Fanuc TP program (LS listing): UP025.LS

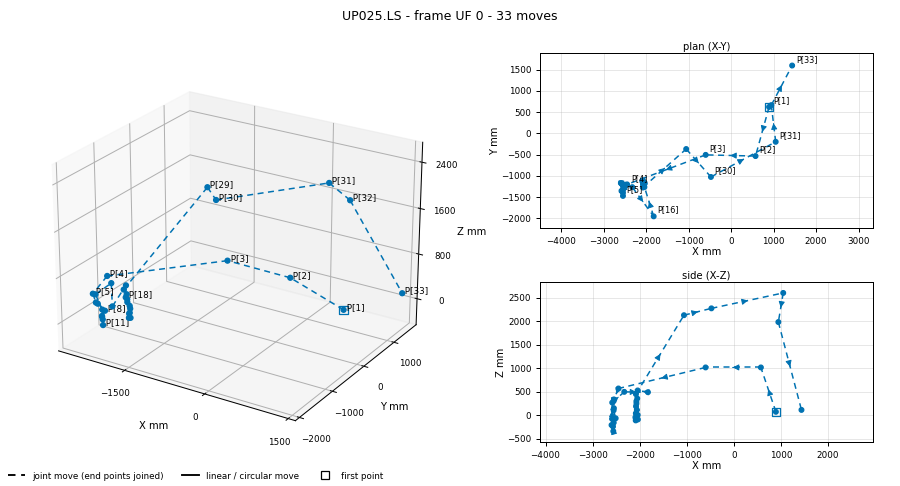
[picture p0: tool path of UP025.LS in frame UF 0, 33 of 33 moves have a stored position in this frame; points joined in program order, loops and branches not executed]
/PROG  UP025
/ATTR
OWNER		= GME;
COMMENT		= "DEPOSITA ST1150";
PROG_SIZE	= 15100;
CREATE		= DATE 03-01-27  TIME 10:40:16;
MODIFIED	= DATE 24-05-04  TIME 16:17:32;
FILE_NAME	= UP025;
VERSION		= 0;
LINE_COUNT	= 60;
MEMORY_SIZE	= 27460;
PROTECT		= READ_WRITE;
TCD:  STACK_SIZE	= 500,
      TASK_PRIORITY	= 50,
      TIME_SLICE	= 0,
      BUSY_LAMP_OFF	= 0,
      ABORT_REQUEST	= 0,
      PAUSE_REQUEST	= 0;
DEFAULT_GROUP	= 1,1,1,1,*;
CONTROL_CODE	= 00000000 00000000;
/APPL
/MN
   1:  UFRAME_NUM=0 ;
   2:  UTOOL_NUM=1 ;
   3:  PAYLOAD[2] ;
   4:  !Apagar Perfil Lib. 74 vs ST1150 ;
   5:  !Apagar Perfil Lib. 73 vs ST1150 ;
   6:  !Encender Anticol. 3 vs 1150R01 ;
   7:  !Encender Anticol. 5 vs 1180R01 ;
   8:J P[1] 100% CNT0 ACC100 TB    0.00sec,P-SPS    ;
      1:  TC_ONLINE (ON) ;
      2:  DO[23]=OFF ;
      3:  TIMER[6]=RESET ;
      4:  TIMER[6]=START ;
      5:  CALL MAKRO050    ;
      6:  !Lib. de Herramientas ;
      7:  DO[80]=ON ;
      8:  DO[78]=OFF ;
      9:  DO[77]=ON ;
     10:  DO[75]=OFF ;
     11:  DO[74]=ON ;
     12:  DO[73]=ON ;
     13:  DO[71]=OFF ;
     14:  DO[70]=OFF ;
     15:  DO[69]=OFF ;
     16:  DO[68]=OFF ;
     17:  DO[67]=OFF ;
     18:  !Lib. de Anticolisiones ;
     19:  DO[41]=ON ;
     20:  DO[42]=ON ;
     21:  DO[43]=ON ;
     22:  DO[44]=ON ;
     23:  DO[45]=ON ;
     24:  DO[46]=ON ;
     25:  !Apagar Pos. Base ;
     26:  DO[15]=OFF ;
     27:  !Robot en Trayectoria ;
     28:  DO[16]=ON ;
     29:  WAIT (DI[74] AND DI[73] AND M[10])    ;
     30:  DO[74]=OFF ;
     31:  DO[73]=OFF ;
     32:  !Encender Anticolisiones ;
     33:  DO[83]=ON ;
     34:  DO[85]=ON ;
     35:  CALL MAKRO020    ;
     36:  WAIT (DI[23])    ;
     37:  DO[23]=ON ;
     38:  !Marcas de Usuario: ;
     39:  !Marca 1 ST1150 Vacia ;
     40:  !M[10]=(!DI[60] AND DI[59] ;
     41:  !AND !DI[58] AND DI[57]) ;
     42:  !Marca 7 Estado de Garra ;
     43:  !Valvula 1,2,3&5 en V, 4,6&7 en R ;
     44:  !M[23]=(M[32] AND M[36] AND M[37] ;
     45:  !AND M[40] AND M[41] AND M[43] ;
     46:  !AND M[63]) ;
     47:  TC_ONLINE (DI[43] AND DI[45] AND DI[73] AND DI[74] AND M[1] AND M[10] AND M[23] AND M[30] AND M[95] AND M[96]) ;
       ------ ;
   9:J P[2] 100% CNT100 ACC100 TB   0.00sec,P-SPS    ;
      1:  TC_ONLINE (DI[43] AND DI[45] AND DI[73] AND DI[74] AND M[1] AND M[10] AND M[23] AND M[30] AND M[95] AND M[96]) ;
       ------ ;
  10:J P[3] 100% CNT100 ACC100 TB   0.00sec,P-SPS    ;
      1:  TC_ONLINE (DI[43] AND DI[45] AND DI[73] AND DI[74] AND M[1] AND M[10] AND M[23] AND M[30] AND M[95] AND M[96]) ;
       ------ ;
  11:J P[4] 100% CNT100 ACC100 TB   0.00sec,P-SPS    ;
      1:  TC_ONLINE (DI[43] AND DI[45] AND DI[73] AND DI[74] AND M[1] AND M[10] AND M[23] AND M[30] AND M[95] AND M[96]) ;
       ------ ;
  12:J P[5] 100% CNT100 ACC100 TB   0.00sec,P-SPS    ;
      1:  TC_ONLINE (DI[43] AND DI[45] AND DI[73] AND DI[74] AND M[1] AND M[10] AND M[23] AND M[30] AND M[95] AND M[96]) ;
       ------ ;
  13:J P[6] 100% CNT100 ACC100 TB   0.00sec,P-SPS    ;
      1:  TC_ONLINE (DI[43] AND DI[45] AND DI[73] AND DI[74] AND M[1] AND M[10] AND M[23] AND M[30] AND M[95] AND M[96]) ;
       ------ ;
  14:J P[7] 100% CNT100 ACC100 TB   0.00sec,P-SPS    ;
      1:  TC_ONLINE (DI[43] AND DI[45] AND DI[73] AND DI[74] AND M[1] AND M[10] AND M[23] AND M[30] AND M[95] AND M[96]) ;
       ------ ;
  15:J P[8] 100% CNT100 ACC100 TB   0.00sec,P-SPS    ;
      1:  TC_ONLINE (DI[43] AND DI[45] AND DI[73] AND DI[74] AND M[1] AND M[10] AND M[23] AND M[30] AND M[95] AND M[96]) ;
       ------ ;
  16:J P[9] 100% CNT100 ACC100 TB   0.00sec,P-SPS    ;
      1:  TC_ONLINE (DI[43] AND DI[45] AND DI[73] AND DI[74] AND M[1] AND M[10] AND M[23] AND M[30] AND M[95] AND M[96]) ;
       ------ ;
  17:J P[10] 100% CNT0 ACC100 TB    .10sec,P-SPS    ;
      1:  TC_ONLINE (ON) ;
      2:  DO[23]=OFF ;
      3:  F[6]=(ON) ;
      4:  CALL MAKRO343    ;
      5:  WAIT (M[42])    ;
      6:  WAIT (DI[23])    ;
      7:  DO[23]=ON ;
      8:  !Marca 8 Estado de Garra ;
      9:  !Valvula 1,2,3,5&6 en V, 4&7 en R ;
     10:  !M[24]=(M[32] AND M[36] AND M[37] ;
     11:  !AND M[40] AND M[42] AND M[43] ;
     12:  !AND M[63]) ;
     13:  TC_ONLINE (DI[43] AND DI[45] AND DI[73] AND DI[74] AND M[1] AND M[24] AND M[30] AND M[95] AND M[96]) ;
       ------ ;
  18:   ;
  19:  !En Posicion 1 ST1150 ;
  20:  !Dejar Pieza 1 en ST1150 ;
  21:  !Fin de Trabajo 4 ;
  22:L P[11] 1500mm/sec CNT0 ACC100 TB    .10sec,P-SPS    ;
      1:  TC_ONLINE (ON) ;
      2:  DO[23]=OFF ;
      3:  WAIT ((!DI[59] AND DI[60]) OR DI[15])    ;
      4:  F[1]=(ON) ;
      5:  CALL MAKRO342    ;
      6:  CALL MAKRO340    ;
      7:  WAIT (M[31])    ;
      8:  DO[71]=ON ;
      9:  CALL MAKRO004    ;
     10:  WAIT (DI[72])    ;
     11:  DO[71]=OFF ;
     12:  WAIT (DI[23])    ;
     13:  DO[23]=ON ;
     14:  !Marca 2 ST1150 C/Pieza 1 ;
     15:  !M[11]=(DI[60] AND !DI[59] ;
     16:  !AND !DI[58] AND DI[57]) ;
     17:  !Marca 9 Estado de Garra ;
     18:  !Valvula 2,3,5&6 en V, 1,4&7 en R ;
     19:  !M[25]=(M[31] AND M[36] AND M[37] ;
     20:  !AND M[40] AND M[42] AND M[43] ;
     21:  !AND M[63]) ;
     22:  TC_ONLINE (DI[43] AND DI[45] AND DI[72] AND DI[74] AND M[11] AND M[25] AND M[30] AND M[95] AND M[96]) ;
       ------ ;
  23:   ;
  24:L P[12] 2000mm/sec CNT0 ACC100 TB    .10sec,P-SPS    ;
      1:  TC_ONLINE (ON) ;
      2:  DO[23]=OFF ;
      3:  WAIT (M[5])    ;
      4:  WAIT (DI[23])    ;
      5:  DO[23]=ON ;
      6:  TC_ONLINE (DI[43] AND DI[45] AND DI[72] AND DI[74] AND M[5] AND M[11] AND M[25] AND M[30] AND M[95] AND M[96]) ;
       ------ ;
  25:   ;
  26:J P[13] 100% CNT100 ACC100 TB   0.00sec,P-SPS    ;
      1:  TC_ONLINE (DI[43] AND DI[45] AND DI[72] AND DI[74] AND M[5] AND M[11] AND M[25] AND M[30] AND M[95] AND M[96]) ;
       ------ ;
  27:J P[14] 100% CNT100 ACC100 TB   0.00sec,P-SPS    ;
      1:  TC_ONLINE (DI[43] AND DI[45] AND DI[72] AND DI[74] AND M[5] AND M[11] AND M[25] AND M[30] AND M[95] AND M[96]) ;
       ------ ;
  28:J P[15] 100% CNT100 ACC100 TB   0.00sec,P-SPS    ;
      1:  TC_ONLINE (DI[43] AND DI[45] AND DI[72] AND DI[74] AND M[5] AND M[11] AND M[25] AND M[30] AND M[95] AND M[96]) ;
       ------ ;
  29:J P[16] 100% CNT100 ACC100 TB   0.00sec,P-SPS    ;
      1:  TC_ONLINE (DI[43] AND DI[45] AND DI[72] AND DI[74] AND M[5] AND M[11] AND M[25] AND M[30] AND M[95] AND M[96]) ;
       ------ ;
  30:  UTOOL_NUM=2 ;
  31:J P[17] 100% CNT0 ACC100 TB    .10sec,P-SPS    ;
      1:  TC_ONLINE (ON) ;
      2:  DO[23]=OFF ;
      3:  DO[70]=ON ;
      4:  WAIT (DI[70])    ;
      5:  DO[70]=OFF ;
      6:  WAIT (DI[23])    ;
      7:  DO[23]=ON ;
      8:  TC_ONLINE (DI[43] AND DI[45] AND DI[70] AND DI[74] AND M[5] AND M[11] AND M[25] AND M[30] AND M[95] AND M[96]) ;
       ------ ;
  32:J P[18] 100% CNT100 ACC100 TB   0.00sec,P-SPS    ;
      1:  TC_ONLINE (DI[43] AND DI[45] AND DI[70] AND DI[74] AND M[5] AND M[11] AND M[25] AND M[30] AND M[95] AND M[96]) ;
       ------ ;
  33:J P[19] 100% CNT100 ACC100 TB   0.00sec,P-SPS    ;
      1:  TC_ONLINE (DI[43] AND DI[45] AND DI[70] AND DI[74] AND M[5] AND M[11] AND M[25] AND M[30] AND M[95] AND M[96]) ;
       ------ ;
  34:J P[20] 100% CNT100 ACC100 TB   0.00sec,P-SPS    ;
      1:  TC_ONLINE (DI[43] AND DI[45] AND DI[70] AND DI[74] AND M[5] AND M[11] AND M[25] AND M[30] AND M[95] AND M[96]) ;
       ------ ;
  35:J P[21] 100% CNT100 ACC100 TB   0.00sec,P-SPS    ;
      1:  TC_ONLINE (DI[43] AND DI[45] AND DI[70] AND DI[74] AND M[5] AND M[25] AND M[30] AND M[95] AND M[96]) ;
       ------ ;
  36:J P[22] 100% CNT0 ACC100 TB    .10sec,P-SPS    ;
      1:  TC_ONLINE (ON) ;
      2:  DO[23]=(OFF) ;
      3:  WAIT (DI[23])    ;
      4:  DO[23]=(ON) ;
      5:  TC_ONLINE (DI[43] AND DI[45] AND DI[70] AND DI[74] AND M[5] AND M[25] AND M[30] AND M[95] AND M[96]) ;
       ------ ;
  37:J P[23] 100% CNT0 ACC100 TB    .10sec,P-SPS    ;
      1:  TC_ONLINE (ON) ;
      2:  DO[23]=(OFF) ;
      3:  WAIT (DI[23])    ;
      4:  DO[23]=(ON) ;
      5:  TC_ONLINE (DI[43] AND DI[45] AND DI[70] AND DI[74] AND M[5] AND M[25] AND M[30] AND M[95] AND M[96]) ;
       ------ ;
  38:   ;
  39:  !En Posicion 2 ST1150 ;
  40:  !Dejar Pieza 2 en ST1150 ;
  41:  !Fin de Trabajo 5 ;
  42:L P[24] 1500mm/sec CNT0 ACC100 TB    .10sec,P-SPS    ;
      1:  TC_ONLINE (ON) ;
      2:  DO[23]=OFF ;
      3:  DO[68]=ON ;
      4:  WAIT ((!DI[57] AND DI[58]) OR DI[15])    ;
      5:  F[3]=(ON) ;
      6:  CALL MAKRO342    ;
      7:  CALL MAKRO340    ;
      8:  WAIT (M[35])    ;
      9:  F[7]=(ON) ;
     10:  CALL MAKRO343    ;
     11:  WAIT (M[44])    ;
     12:  DO[69]=ON ;
     13:  CALL MAKRO005    ;
     14:  WAIT (DI[69])    ;
     15:  DO[69]=OFF ;
     16:  F[5]=(ON) ;
     17:  CALL MAKRO342    ;
     18:  CALL MAKRO340    ;
     19:  WAIT (M[39])    ;
     20:  F[4]=(ON) ;
     21:  CALL MAKRO343    ;
     22:  WAIT (M[38])    ;
     23:  DO[67]=(ON) ;
     24:  WAIT (DI[67])    ;
     25:  DO[67]=(OFF) ;
     26:  IF (!DI[15]),F[17]=(ON) ;
     27:  IF (!DI[15]),CALL MAKRO342 ;
     28:  CALL MAKRO340    ;
     29:  WAIT (!M[63] OR M[63] OR DI[15])    ;
     30:  F[7]=(ON) ;
     31:  CALL MAKRO342    ;
     32:  CALL MAKRO340    ;
     33:  WAIT (M[43])    ;
     34:  WAIT (DI[23])    ;
     35:  DO[23]=ON ;
     36:  !Marca 3 ST1150 Llena ;
     37:  !M[12]=(DI[60] AND !DI[59] ;
     38:  !AND DI[58] AND !DI[57]) ;
     39:  !Marca 10 Estado de Garra ;
     40:  !Valvula 4&6 en V, 1,2,3,5&7 en R ;
     41:  !M[26]=(M[31] AND M[35] AND M[38] ;
     42:  !AND M[39] AND M[42] AND M[43]) ;
     43:  TC_ONLINE (DI[43] AND DI[45] AND DI[67] AND DI[74] AND M[12] AND M[26] AND M[30] AND M[95] AND M[96]) ;
       ------ ;
  43:   ;
  44:  PAYLOAD[1] ;
  45:L P[25] 2000mm/sec CNT0 ACC100 TB    .10sec,P-SPS    ;
      1:  TC_ONLINE (ON) ;
      2:  DO[23]=OFF ;
      3:  WAIT (DI[23])    ;
      4:  DO[23]=ON ;
      5:  TC_ONLINE (DI[43] AND DI[45] AND DI[67] AND DI[74] AND M[12] AND M[26] AND M[30] AND M[95] AND M[96]) ;
       ------ ;
  46:J P[26] 100% CNT100 ACC100 TB   0.00sec,P-SPS    ;
      1:  TC_ONLINE (DI[43] AND DI[45] AND DI[67] AND DI[74] AND M[12] AND M[26] AND M[30] AND M[95] AND M[96]) ;
       ------ ;
  47:J P[27] 100% CNT100 ACC100 TB   0.00sec,P-SPS    ;
      1:  TC_ONLINE (DI[43] AND DI[45] AND DI[67] AND DI[74] AND M[12] AND M[26] AND M[30] AND M[95] AND M[96]) ;
       ------ ;
  48:   ;
  49:J P[28] 100% CNT100 ACC100 TB   0.00sec,P-SPS    ;
      1:  TC_ONLINE (DI[43] AND DI[45] AND DI[67] AND DI[74] AND M[2] AND M[12] AND M[26] AND M[30] AND M[95] AND M[96]) ;
       ------ ;
  50:   ;
  51:  !Encender Perfil Lib 73 vs ST1150 ;
  52:J P[29] 100% CNT100 ACC100 TB   0.00sec,P-SPS    ;
      1:  TC_ONLINE (ON) ;
      2:  DO[73]=ON ;
      3:  TC_ONLINE (DI[43] AND DI[45] AND DI[74] AND M[2] AND M[12] AND M[26] AND M[30] AND M[95] AND M[96]) ;
       ------ ;
  53:   ;
  54:  !Encender Perfil Lib 74 vs ST1150 ;
  55:  !Apagar Anticol. 3 vs 1150R01 ;
  56:  !Apagar Anticol. 5 vs 1180R01 ;
  57:J P[30] 100% CNT100 ACC100 TB   0.00sec,P-SPS    ;
      1:  TC_ONLINE (ON) ;
      2:  DO[74]=ON ;
      3:  DO[43]=ON ;
      4:  DO[45]=ON ;
      5:  TC_ONLINE (M[2] AND M[26] AND M[30] AND M[95] AND M[96]) ;
       ------ ;
  58:J P[31] 100% CNT100 ACC100 TB   0.00sec,P-SPS    ;
      1:  TC_ONLINE (M[2] AND M[26] AND M[30] AND M[95] AND M[96]) ;
       ------ ;
  59:J P[32] 100% CNT100 ACC100 TB   0.00sec,P-SPS    ;
      1:  TC_ONLINE (M[2] AND M[26] AND M[30] AND M[95] AND M[96]) ;
       ------ ;
  60:J P[33] 100% CNT0 ACC100 TB    .10sec,P-SPS    ;
      1:  TC_ONLINE (ON) ;
      2:  DO[23]=OFF ;
      3:  TIMER[6]=STOP ;
      4:  F[4]=(ON) ;
      5:  F[6]=(ON) ;
      6:  CALL MAKRO342    ;
      7:  CALL MAKRO340    ;
      8:  WAIT (M[37] AND M[41])    ;
      9:  WAIT (DI[23])    ;
     10:  DO[23]=ON ;
     11:  !Marca 4 Estado de Garra ;
     12:  !Valvulas 1-7 en R ;
     13:  !M[20]=(M[31] AND M[35] AND M[37] ;
     14:  !AND M[39] AND M[41] AND M[43]) ;
     15:  TC_ONLINE (M[20] AND M[2] AND M[30] AND M[95] AND M[96]) ;
       ------ ;
/POS
P[1]{
   GP1:
	UF : 0, UT : 1,		CONFIG : 'N U T, 0, 0, 0',
	X =   893.302  mm,	Y =   623.420  mm,	Z =    77.203  mm,
	W =    98.852 deg,	P =    39.834 deg,	R =  -104.177 deg
   GP2:
	UF : 0, UT : 1,
	J1=   100.000  mm
   GP3:
	UF : 0, UT : 1,
	J1=     0.000  mm
   GP4:
	UF : 0, UT : 1,
	J1=     0.000  mm
};
P[2]{
   GP1:
	UF : 0, UT : 1,		CONFIG : 'N U T, 0, 0, 0',
	X =   574.660  mm,	Y =  -533.643  mm,	Z =  1020.134  mm,
	W =  -149.104 deg,	P =    53.651 deg,	R =   -86.456 deg
   GP2:
	UF : 0, UT : 1,
	J1=   100.000  mm
   GP3:
	UF : 0, UT : 1,
	J1=     0.000  mm
   GP4:
	UF : 0, UT : 1,
	J1=     0.000  mm
};
P[3]{
   GP1:
	UF : 0, UT : 1,		CONFIG : 'N U T, 0, 0, 0',
	X =  -599.745  mm,	Y =  -505.284  mm,	Z =  1020.134  mm,
	W =  -149.104 deg,	P =    53.651 deg,	R =   176.539 deg
   GP2:
	UF : 0, UT : 1,
	J1=   100.000  mm
   GP3:
	UF : 0, UT : 1,
	J1=     0.000  mm
   GP4:
	UF : 0, UT : 1,
	J1=     0.000  mm
};
P[4]{
   GP1:
	UF : 0, UT : 1,		CONFIG : 'N U T, 0, 0, 0',
	X = -2450.973  mm,	Y = -1200.381  mm,	Z =   572.809  mm,
	W =    13.060 deg,	P =    75.060 deg,	R =  -149.650 deg
   GP2:
	UF : 0, UT : 1,
	J1=   100.000  mm
   GP3:
	UF : 0, UT : 1,
	J1=     0.000  mm
   GP4:
	UF : 0, UT : 1,
	J1=     0.000  mm
};
P[5]{
   GP1:
	UF : 0, UT : 1,		CONFIG : 'N U T, 0, 0, 0',
	X = -2547.951  mm,	Y = -1471.892  mm,	Z =   341.201  mm,
	W =     1.514 deg,	P =    73.231 deg,	R =  -148.514 deg
   GP2:
	UF : 0, UT : 1,
	J1=   100.000  mm
   GP3:
	UF : 0, UT : 1,
	J1=     0.000  mm
   GP4:
	UF : 0, UT : 1,
	J1=     0.000  mm
};
P[6]{
   GP1:
	UF : 0, UT : 1,		CONFIG : 'N U T, 0, 0, 0',
	X = -2547.909  mm,	Y = -1396.949  mm,	Z =   154.448  mm,
	W =      .893 deg,	P =    75.485 deg,	R =  -149.123 deg
   GP2:
	UF : 0, UT : 1,
	J1=   100.000  mm
   GP3:
	UF : 0, UT : 1,
	J1=     0.000  mm
   GP4:
	UF : 0, UT : 1,
	J1=     0.000  mm
};
P[7]{
   GP1:
	UF : 0, UT : 1,		CONFIG : 'N U T, 0, 0, 0',
	X = -2553.313  mm,	Y = -1338.897  mm,	Z =   109.022  mm,
	W =      .420 deg,	P =    77.991 deg,	R =  -153.363 deg
   GP2:
	UF : 0, UT : 1,
	J1=   100.000  mm
   GP3:
	UF : 0, UT : 1,
	J1=     0.000  mm
   GP4:
	UF : 0, UT : 1,
	J1=     0.000  mm
};
P[8]{
   GP1:
	UF : 0, UT : 1,		CONFIG : 'N U T, 0, 0, 0',
	X = -2509.638  mm,	Y = -1206.159  mm,	Z =   -60.188  mm,
	W =     -.006 deg,	P =    84.228 deg,	R =  -150.013 deg
   GP2:
	UF : 0, UT : 1,
	J1=   100.000  mm
   GP3:
	UF : 0, UT : 1,
	J1=     0.000  mm
   GP4:
	UF : 0, UT : 1,
	J1=     0.000  mm
};
P[9]{
   GP1:
	UF : 0, UT : 1,		CONFIG : 'N U T, 0, 0, 0',
	X = -2550.680  mm,	Y = -1236.247  mm,	Z =  -152.696  mm,
	W =     -.007 deg,	P =    84.227 deg,	R =  -150.012 deg
   GP2:
	UF : 0, UT : 1,
	J1=   100.000  mm
   GP3:
	UF : 0, UT : 1,
	J1=     0.000  mm
   GP4:
	UF : 0, UT : 1,
	J1=     0.000  mm
};
P[10]{
   GP1:
	UF : 0, UT : 1,		CONFIG : 'N U T, 0, 0, 0',
	X = -2566.540  mm,	Y = -1195.918  mm,	Z =  -235.071  mm,
	W =    -2.590 deg,	P =    85.647 deg,	R =  -152.005 deg
   GP2:
	UF : 0, UT : 1,
	J1=   101.322  mm
   GP3:
	UF : 0, UT : 1,
	J1=     0.000  mm
   GP4:
	UF : 0, UT : 1,
	J1=     0.000  mm
};
P[11]{
   GP1:
	UF : 0, UT : 1,		CONFIG : 'N U T, 0, 0, 0',
	X = -2560.261  mm,	Y = -1200.023  mm,	Z =  -334.405  mm,
	W =    25.250 deg,	P =    87.683 deg,	R =  -124.023 deg
   GP2:
	UF : 0, UT : 1,
	J1=   106.400  mm
   GP3:
	UF : 0, UT : 1,
	J1=     0.000  mm
   GP4:
	UF : 0, UT : 1,
	J1=     0.000  mm
};
P[12]{
   GP1:
	UF : 0, UT : 1,		CONFIG : 'N U T, 0, 0, 0',
	X = -2597.734  mm,	Y = -1168.977  mm,	Z =  -203.862  mm,
	W =     8.862 deg,	P =    86.601 deg,	R =  -141.113 deg
   GP2:
	UF : 0, UT : 1,
	J1=   100.002  mm
   GP3:
	UF : 0, UT : 1,
	J1=     0.000  mm
   GP4:
	UF : 0, UT : 1,
	J1=     0.000  mm
};
P[13]{
   GP1:
	UF : 0, UT : 1,		CONFIG : 'N U T, 0, 0, 0',
	X = -2586.677  mm,	Y = -1173.902  mm,	Z =   -72.188  mm,
	W =      .000 deg,	P =    87.427 deg,	R =  -150.005 deg
   GP2:
	UF : 0, UT : 1,
	J1=   100.002  mm
   GP3:
	UF : 0, UT : 1,
	J1=     0.000  mm
   GP4:
	UF : 0, UT : 1,
	J1=     0.000  mm
};
P[14]{
   GP1:
	UF : 0, UT : 1,		CONFIG : 'N U T, 0, 0, 0',
	X = -2582.668  mm,	Y = -1353.251  mm,	Z =   273.693  mm,
	W =   -20.996 deg,	P =    72.024 deg,	R =  -171.741 deg
   GP2:
	UF : 0, UT : 1,
	J1=   100.000  mm
   GP3:
	UF : 0, UT : 1,
	J1=     0.000  mm
   GP4:
	UF : 0, UT : 1,
	J1=     0.000  mm
};
P[15]{
   GP1:
	UF : 0, UT : 1,		CONFIG : 'N U T, 0, 0, 0',
	X = -2327.345  mm,	Y = -1265.489  mm,	Z =   501.373  mm,
	W =     1.785 deg,	P =    73.144 deg,	R =  -148.053 deg
   GP2:
	UF : 0, UT : 1,
	J1=   100.000  mm
   GP3:
	UF : 0, UT : 1,
	J1=     0.000  mm
   GP4:
	UF : 0, UT : 1,
	J1=     0.000  mm
};
P[16]{
   GP1:
	UF : 0, UT : 1,		CONFIG : 'N U T, 0, 0, 0',
	X = -1824.464  mm,	Y = -1953.321  mm,	Z =   494.068  mm,
	W =    37.586 deg,	P =    69.200 deg,	R =  -102.660 deg
   GP2:
	UF : 0, UT : 1,
	J1=   100.000  mm
   GP3:
	UF : 0, UT : 1,
	J1=     0.000  mm
   GP4:
	UF : 0, UT : 1,
	J1=     0.000  mm
};
P[17]{
   GP1:
	UF : 0, UT : 2,		CONFIG : 'N U T, 0, 0, 0',
	X = -2042.524  mm,	Y = -1262.616  mm,	Z =   531.178  mm,
	W =   -22.630 deg,	P =    84.645 deg,	R =  -169.649 deg
   GP2:
	UF : 0, UT : 2,
	J1=   100.000  mm
   GP3:
	UF : 0, UT : 2,
	J1=     0.000  mm
   GP4:
	UF : 0, UT : 2,
	J1=     0.000  mm
};
P[18]{
   GP1:
	UF : 0, UT : 2,		CONFIG : 'N U T, 0, 0, 0',
	X = -2070.063  mm,	Y = -1237.595  mm,	Z =   302.228  mm,
	W =   -55.461 deg,	P =    86.280 deg,	R =   152.256 deg
   GP2:
	UF : 0, UT : 2,
	J1=   100.000  mm
   GP3:
	UF : 0, UT : 2,
	J1=     0.000  mm
   GP4:
	UF : 0, UT : 2,
	J1=     0.000  mm
};
P[19]{
   GP1:
	UF : 0, UT : 2,		CONFIG : 'N U T, 0, 0, 0',
	X = -2068.144  mm,	Y = -1200.037  mm,	Z =   253.507  mm,
	W =   -55.461 deg,	P =    86.280 deg,	R =   152.256 deg
   GP2:
	UF : 0, UT : 2,
	J1=   100.000  mm
   GP3:
	UF : 0, UT : 2,
	J1=     0.000  mm
   GP4:
	UF : 0, UT : 2,
	J1=     0.000  mm
};
P[20]{
   GP1:
	UF : 0, UT : 2,		CONFIG : 'N U T, 0, 0, 0',
	X = -2077.670  mm,	Y = -1185.065  mm,	Z =   194.148  mm,
	W =   -86.617 deg,	P =    86.322 deg,	R =   124.811 deg
   GP2:
	UF : 0, UT : 2,
	J1=   100.000  mm
   GP3:
	UF : 0, UT : 2,
	J1=     0.000  mm
   GP4:
	UF : 0, UT : 2,
	J1=     0.000  mm
};
P[21]{
   GP1:
	UF : 0, UT : 2,		CONFIG : 'N U T, 0, 0, 0',
	X = -2081.543  mm,	Y = -1103.385  mm,	Z =    44.980  mm,
	W =   -92.311 deg,	P =    86.253 deg,	R =   113.508 deg
   GP2:
	UF : 0, UT : 2,
	J1=   101.800  mm
   GP3:
	UF : 0, UT : 2,
	J1=     0.000  mm
   GP4:
	UF : 0, UT : 2,
	J1=     0.000  mm
};
P[22]{
   GP1:
	UF : 0, UT : 2,		CONFIG : 'N U T, 0, 0, 0',
	X = -2091.079  mm,	Y = -1121.986  mm,	Z =   -40.034  mm,
	W =   -88.730 deg,	P =    86.241 deg,	R =   120.751 deg
   GP2:
	UF : 0, UT : 2,
	J1=   100.000  mm
   GP3:
	UF : 0, UT : 2,
	J1=     0.000  mm
   GP4:
	UF : 0, UT : 2,
	J1=     0.000  mm
};
P[23]{
   GP1:
	UF : 0, UT : 2,		CONFIG : 'N U T, 0, 0, 0',
	X = -2084.259  mm,	Y = -1140.649  mm,	Z =  -105.346  mm,
	W =  -102.582 deg,	P =    85.651 deg,	R =   108.498 deg
   GP2:
	UF : 0, UT : 2,
	J1=   100.300  mm
   GP3:
	UF : 0, UT : 2,
	J1=     0.000  mm
   GP4:
	UF : 0, UT : 2,
	J1=     0.000  mm
};
P[24]{
   GP1:
	UF : 0, UT : 2,		CONFIG : 'N U T, 0, 0, 0',
	X = -2038.457  mm,	Y = -1161.573  mm,	Z =   -85.450  mm,
	W =   -96.937 deg,	P =    85.752 deg,	R =   113.846 deg
   GP2:
	UF : 0, UT : 2,
	J1=   125.900  mm
   GP3:
	UF : 0, UT : 2,
	J1=     0.000  mm
   GP4:
	UF : 0, UT : 2,
	J1=     0.000  mm
};
P[25]{
   GP1:
	UF : 0, UT : 2,		CONFIG : 'N U T, 0, 0, 0',
	X = -2041.928  mm,	Y = -1176.308  mm,	Z =    10.928  mm,
	W =   -97.744 deg,	P =    85.754 deg,	R =   113.916 deg
   GP2:
	UF : 0, UT : 2,
	J1=   122.300  mm
   GP3:
	UF : 0, UT : 2,
	J1=     0.000  mm
   GP4:
	UF : 0, UT : 2,
	J1=     0.000  mm
};
P[26]{
   GP1:
	UF : 0, UT : 2,		CONFIG : 'N U T, 0, 0, 0',
	X = -2060.172  mm,	Y = -1146.796  mm,	Z =   116.923  mm,
	W =  -100.313 deg,	P =    85.837 deg,	R =   111.083 deg
   GP2:
	UF : 0, UT : 2,
	J1=   100.000  mm
   GP3:
	UF : 0, UT : 2,
	J1=     0.000  mm
   GP4:
	UF : 0, UT : 2,
	J1=     0.000  mm
};
P[27]{
   GP1:
	UF : 0, UT : 2,		CONFIG : 'N U T, 0, 0, 0',
	X = -2051.278  mm,	Y = -1235.471  mm,	Z =   361.272  mm,
	W =   -88.707 deg,	P =    86.138 deg,	R =   123.884 deg
   GP2:
	UF : 0, UT : 2,
	J1=   100.000  mm
   GP3:
	UF : 0, UT : 2,
	J1=     0.000  mm
   GP4:
	UF : 0, UT : 2,
	J1=     0.000  mm
};
P[28]{
   GP1:
	UF : 0, UT : 2,		CONFIG : 'N U T, 0, 0, 0',
	X = -2079.395  mm,	Y = -1274.561  mm,	Z =   452.593  mm,
	W =   -83.942 deg,	P =    86.190 deg,	R =   129.109 deg
   GP2:
	UF : 0, UT : 2,
	J1=   100.000  mm
   GP3:
	UF : 0, UT : 2,
	J1=     0.000  mm
   GP4:
	UF : 0, UT : 2,
	J1=     0.000  mm
};
P[29]{
   GP1:
	UF : 0, UT : 2,		CONFIG : 'N U T, 0, 0, 0',
	X = -1058.805  mm,	Y =  -367.660  mm,	Z =  2129.829  mm,
	W =     3.506 deg,	P =    27.246 deg,	R =  -145.763 deg
   GP2:
	UF : 0, UT : 2,
	J1=   100.000  mm
   GP3:
	UF : 0, UT : 2,
	J1=     0.000  mm
   GP4:
	UF : 0, UT : 2,
	J1=     0.000  mm
};
P[30]{
   GP1:
	UF : 0, UT : 2,		CONFIG : 'N U T, 0, 0, 0',
	X =  -475.910  mm,	Y = -1025.833  mm,	Z =  2275.270  mm,
	W =     4.453 deg,	P =    17.669 deg,	R =   -99.640 deg
   GP2:
	UF : 0, UT : 2,
	J1=   100.000  mm
   GP3:
	UF : 0, UT : 2,
	J1=     0.000  mm
   GP4:
	UF : 0, UT : 2,
	J1=     0.000  mm
};
P[31]{
   GP1:
	UF : 0, UT : 2,		CONFIG : 'N U T, 0, 0, 0',
	X =  1049.266  mm,	Y =  -197.396  mm,	Z =  2602.499  mm,
	W =     6.406 deg,	P =    -4.413 deg,	R =     6.057 deg
   GP2:
	UF : 0, UT : 2,
	J1=   100.000  mm
   GP3:
	UF : 0, UT : 2,
	J1=     0.000  mm
   GP4:
	UF : 0, UT : 2,
	J1=     0.000  mm
};
P[32]{
   GP1:
	UF : 0, UT : 2,		CONFIG : 'N U T, 0, 0, 0',
	X =   945.887  mm,	Y =   665.819  mm,	Z =  1984.355  mm,
	W =  -124.411 deg,	P =    15.627 deg,	R =    12.586 deg
   GP2:
	UF : 0, UT : 2,
	J1=   100.000  mm
   GP3:
	UF : 0, UT : 2,
	J1=     0.000  mm
   GP4:
	UF : 0, UT : 2,
	J1=     0.000  mm
};
P[33]{
   GP1:
	UF : 0, UT : 2,		CONFIG : 'N U T, 0, 0, 0',
	X =  1436.857  mm,	Y =  1598.998  mm,	Z =   117.965  mm,
	W =   179.395 deg,	P =    81.558 deg,	R =   -18.495 deg
   GP2:
	UF : 0, UT : 2,
	J1=   100.000  mm
   GP3:
	UF : 0, UT : 2,
	J1=     0.000  mm
   GP4:
	UF : 0, UT : 2,
	J1=     0.000  mm
};
/END
